FUNCTION_BLOCK SUBSCRIBE_10 (* Subscribe to a PUBLISH_10 Block *)
  (* Description: Copyright (c) 2017 fortiss GmbH This program and the accompanying materials are made available under the terms of the Eclipse Public License 2.0 which is available at https://www.eclipse.org/legal/epl-2.0/ SPDX-License-Identifier: EPL-2.0 *)
  (* Version 1.0, 2017-10-25, Alois Zoitl, fortiss GmbH, initial API and implementation and/or initial documentation *)
  {SET_ATTRIBUTE(GenericClassName, 'GEN_SUBSCRIBE')}
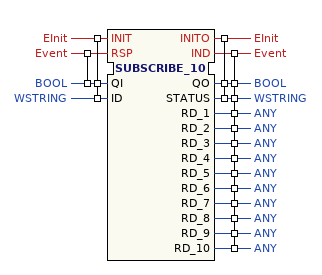
  EVENT_INPUT
    INIT : EInit WITH QI, ID;
    RSP WITH QI;
  END_EVENT
  EVENT_OUTPUT
    INITO : EInit WITH QO, STATUS;
    IND WITH QO, STATUS, RD_1, RD_3, RD_2, RD_4, RD_5, RD_6, RD_7, RD_8, RD_9, RD_10; (* New data available *)
  END_EVENT
  VAR_INPUT
    QI : BOOL;
    ID : WSTRING;
  END_VAR
  VAR_OUTPUT
    QO : BOOL;
    STATUS : WSTRING;
    RD_1 : ANY;
    RD_2 : ANY;
    RD_3 : ANY;
    RD_4 : ANY;
    RD_5 : ANY;
    RD_6 : ANY;
    RD_7 : ANY;
    RD_8 : ANY;
    RD_9 : ANY;
    RD_10 : ANY;
  END_VAR
  (* Service APPLICATION/RESOURCE: Subscribe to a PUBLISH_10 Block *)
END_FUNCTION_BLOCK
